FUNCTION_BLOCK RenderRot (* Rendering Image With Rotation *)
  (* Standard: 61499-2 *)
  (* Version 0.2, 2006-01-05, Anirudha, UoA, Added Layer attribute *)
  (* Version 0.1, 2005-12-04, Anirudha, UoA, Added Angle attribute *)
  (* Compiler header: package fb.rt.vhmi; *)
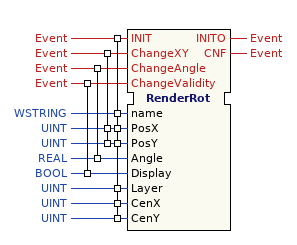
  EVENT_INPUT
    INIT WITH name, PosX, PosY, Layer, CenY, CenX; (* Initialization Request *)
    ChangeXY WITH PosX, PosY; (* Normal Execution Request *)
    ChangeAngle WITH Angle;
    ChangeValidity WITH Display;
  END_EVENT
  EVENT_OUTPUT
    INITO; (* Initialization Confirm *)
    CNF; (* Execution Confirmation *)
  END_EVENT
  VAR_INPUT
    name : WSTRING;
    PosX : UINT;
    PosY : UINT;
    Angle : REAL;
    Display : BOOL;
    Layer : UINT;
    CenX : UINT;
    CenY : UINT;
  END_VAR
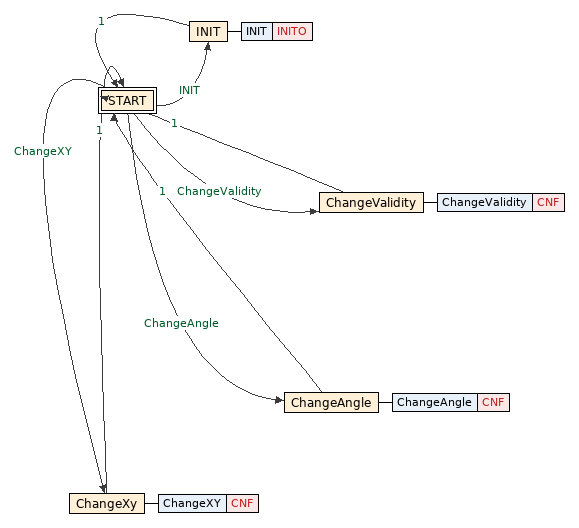
  EC_STATES
    START; (* Initial State *)
    INIT : INIT -> INITO; (* Initialization *)
    ChangeXy : ChangeXY -> CNF;
    ChangeAngle : ChangeAngle -> CNF;
    ChangeValidity : ChangeValidity -> CNF;
  END_STATES
  EC_TRANSITIONS
    START TO INIT := INIT;
    INIT TO START := 1;
    START TO ChangeXy := ChangeXY;
    START TO ChangeAngle := ChangeAngle;
    START TO ChangeValidity := ChangeValidity;
    ChangeXy TO START := 1;
    ChangeAngle TO START := 1;
    ChangeValidity TO START := 1;
  END_TRANSITIONS
  ALGORITHM INIT IN Java: (* Initialization algorithm *)
System.out.print("Name: ");
System.out.println(name.value);
System.out.print("Position: ");
System.out.print(PosX.value);
System.out.print(",");
System.out.print(PosY.value);
ID = ((ImageResource) this.resource).addImage(loadImage(name.value),PosX.value,PosY.value,Layer.value);
((ImageDev) this.getDevice()).frame.repaint();
String abd = "I am " + name.value + " with ID " + ID;
System.out.println(abd);
if (Angle.value != 0)
  service_ChangeAngle(true);
if (Display.value == false)
  service_ChangeValidity(true);
  END_ALGORITHM
  ALGORITHM ChangeXY IN Java:
((SampleFrame)((ImageDev)(this.getDevice())).frame).redrawXY(ID,PosX.value,PosY.value);
  END_ALGORITHM
  ALGORITHM ChangeAngle IN Java:
((SampleFrame)((ImageDev)(this.getDevice())).frame).redrawAngleCenter(ID,Angle.value,(double)CenX.value,(double)CenY.value);
  END_ALGORITHM
  ALGORITHM ChangeValidity IN Java:
((SampleFrame)((ImageDev)(this.getDevice())).frame).setValidity(ID,Display.value);
  END_ALGORITHM
END_FUNCTION_BLOCK
